FUNCTION_BLOCK VCylinderSA (* Composite Function Block Type *)
  (* Standard: 61499-2 *)
  (* Version 0.0, 9/14/2008, Horst Mayer, nxtControl GmbH, template *)
  PACKAGE Main;
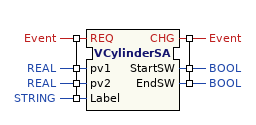
  EVENT_INPUT
    REQ WITH pv1, pv2, Label; (* Normal Execution Request *)
  END_EVENT
  EVENT_OUTPUT
    CHG WITH StartSW, EndSW;
  END_EVENT
  VAR_INPUT
    pv1 : REAL;
    pv2 : REAL;
    Label : STRING;
  END_VAR
  VAR_OUTPUT
    StartSW : BOOL;
    EndSW : BOOL;
  END_VAR
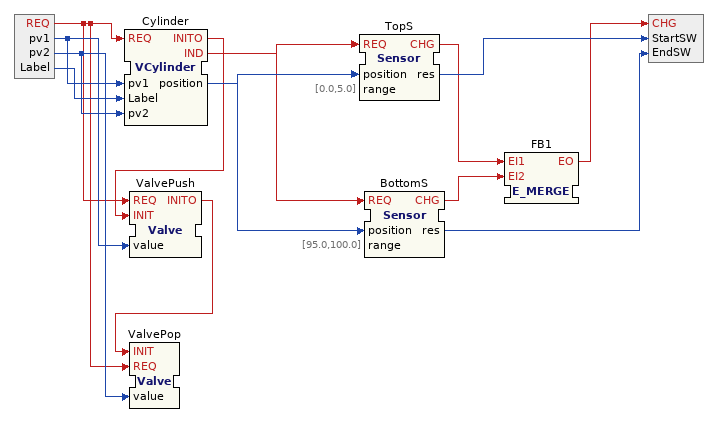
  FBS
    ValvePush : Valve;
    ValvePop : Valve;
    TopS : Sensor(range := [0.0,5.0]);
    BottomS : Sensor(range := [95.0,100.0]);
    FB1 : E_MERGE;
    Cylinder : VCylinder;
  END_FBS
  EVENT_CONNECTIONS
    ValvePush.INITO TO ValvePop.INIT;
    FB1.EO TO CHG;
    REQ TO ValvePush.REQ;
    REQ TO ValvePop.REQ;
    TopS.CHG TO FB1.EI1;
    BottomS.CHG TO FB1.EI2;
    REQ TO Cylinder.REQ;
    Cylinder.INITO TO ValvePush.INIT;
    Cylinder.IND TO TopS.REQ;
    Cylinder.IND TO BottomS.REQ;
  END_CONNECTIONS
  DATA_CONNECTIONS
    TopS.res TO StartSW;
    BottomS.res TO EndSW;
    pv1 TO ValvePush.value;
    pv2 TO ValvePop.value;
    pv1 TO Cylinder.pv1;
    Label TO Cylinder.Label;
    pv2 TO Cylinder.pv2;
    Cylinder.position TO TopS.position;
    Cylinder.position TO BottomS.position;
  END_CONNECTIONS
END_FUNCTION_BLOCK
